// TIA Portal project "MAIN-PLS-AHS-100125" (V19)

(* hardware
DEVICE "S7-1200 station_1"  S7-1200 Station
   slot 0: "Rack_0"  S7-1200 Rack  Rack  V1.0
   slot 1: "PLC_1"  CPU 1214C AC/DC/Rly  6ES7 214-1BG40-0XB0  V4.6
DEVICE "ET 200SP station_1"  ET 200SP-Station
   slot 0: "Rack_0"  Rack  6ES5 710-8MAx1
   slot 0: "et200sp_greider"  IM 155-6 PN HF  6ES7 155-6AU00-0CN0  V4.2
   slot 1: "DI 8x24VDC HF_1"  DI 8x24VDC HF  6ES7 131-6BF00-0CA0  V2.0
      slot 1: "DI 8x24VDC HF_1"  DI 8x24VDC HF
   slot 2: "DI 8x24VDC HF_2"  DI 8x24VDC HF  6ES7 131-6BF00-0CA0  V2.0
      slot 1: "DI 8x24VDC HF_2"  DI 8x24VDC HF
   slot 3: "DI 8x24VDC HF_3"  DI 8x24VDC HF  6ES7 131-6BF00-0CA0  V2.0
      slot 1: "DI 8x24VDC HF_3"  DI 8x24VDC HF
   slot 4: "DI 8x24VDC HF_4"  DI 8x24VDC HF  6ES7 131-6BF00-0CA0  V2.0
      slot 1: "DI 8x24VDC HF_4"  DI 8x24VDC HF
   slot 5: "DQ 8x24VDC/0.5A HF_1"  DQ 8x24VDC/0.5A HF  6ES7 132-6BF00-0CA0  V2.0
      slot 1: "DQ 8x24VDC/0.5A HF_1"  DQ 8x24VDC/0.5A HF
   slot 6: "DQ 8x24VDC/0.5A HF_2"  DQ 8x24VDC/0.5A HF  6ES7 132-6BF00-0CA0  V2.0
      slot 1: "DQ 8x24VDC/0.5A HF_2"  DQ 8x24VDC/0.5A HF
   slot 7: "DQ 8x24VDC/0.5A HF_3"  DQ 8x24VDC/0.5A HF  6ES7 132-6BF00-0CA0  V2.0
      slot 1: "DQ 8x24VDC/0.5A HF_3"  DQ 8x24VDC/0.5A HF
   slot 8: "DQ 8x24VDC/0.5A HF_4"  DQ 8x24VDC/0.5A HF  6ES7 132-6BF00-0CA0  V2.0
      slot 1: "DQ 8x24VDC/0.5A HF_4"  DQ 8x24VDC/0.5A HF
   slot 9: "Server module_1"  Server module  6ES7 193-6PA00-0AA0  V1.1
      slot 1: "Server module_1"  Server module
   slot 127: "BA 2xRJ45"  BA 2xRJ45  6ES7 193-6AR00-0AA0  V0.0
      slot 1: "Port_1"  X1 P1 R  6ES7 193-6AR00-0AA0  V0.0
      slot 2: "Port_2"  X1 P2 R  6ES7 193-6AR00-0AA0  V0.0
DEVICE "ET 200SP station_2"  ET 200SP-Station
   slot 0: "Rack_0"  Rack  6ES5 710-8MAx1
   slot 0: "et200sp_servo"  IM 155-6 PN HF  6ES7 155-6AU00-0CN0  V4.2
   slot 1: "DI 8x24VDC HF_1"  DI 8x24VDC HF  6ES7 131-6BF00-0CA0  V2.0
      slot 1: "DI 8x24VDC HF_1"  DI 8x24VDC HF
   slot 2: "DI 8x24VDC HF_2"  DI 8x24VDC HF  6ES7 131-6BF00-0CA0  V2.0
      slot 1: "DI 8x24VDC HF_2"  DI 8x24VDC HF
   slot 3: "DQ 8x24VDC/0.5A HF_1"  DQ 8x24VDC/0.5A HF  6ES7 132-6BF00-0CA0  V2.0
      slot 1: "DQ 8x24VDC/0.5A HF_1"  DQ 8x24VDC/0.5A HF
   slot 4: "DQ 8x24VDC/0.5A HF_2"  DQ 8x24VDC/0.5A HF  6ES7 132-6BF00-0CA0  V2.0
      slot 1: "DQ 8x24VDC/0.5A HF_2"  DQ 8x24VDC/0.5A HF
   slot 5: "Server module_1"  Server module  6ES7 193-6PA00-0AA0  V1.1
      slot 1: "Server module_1"  Server module
   slot 127: "BA 2xRJ45"  BA 2xRJ45  6ES7 193-6AR00-0AA0  V0.0
      slot 1: "Port_1"  X1 P1 R  6ES7 193-6AR00-0AA0  V0.0
      slot 2: "Port_2"  X1 P2 R  6ES7 193-6AR00-0AA0  V0.0
*)

// ===== PLC "PLC_1"  CPU 1214C AC/DC/Rly =====

VAR_GLOBAL   // PLC tag table "Default tag table"
   "C1.1_I" AT %I2.0 : Bool;
   "C1.2_I" AT %I2.1 : Bool;
   "C2.1_I" AT %I2.2 : Bool;
   "C2.2_I" AT %I2.3 : Bool;
   "C3.1_I" AT %I2.4 : Bool;
   "C3.2_I" AT %I2.5 : Bool;
   "Fotocelle_I" AT %I2.6 : Bool;
   "A_IG_I" AT %I3.1 : Bool;
   "B_IG_I" AT %I3.2 : Bool;
   "Bryter_S1_Ved_HMI_I" AT %I0.0 : Bool;
   "Bryter_S5_Ved_HMI_I" AT %I0.4 : Bool;
   "Bryter_Høyre_Skap_I" AT %I3.3 : Bool;
   "Bryter_Venstre_Skap_I" AT %I3.4 : Bool;
   "Tag_10" AT %IW64 : Word;
   "Bryter_S2_Ved_HMI_I" AT %I0.1 : Bool;
   "Bryter_3_Ved_HMI_I" AT %I0.2 : Bool;
   "Bryter_S4_Ved_HMI_I" AT %I0.3 : Bool;
   "Tag_2" AT %I3.0 : Bool;
   "A-IG" AT %I4.0 : Bool;
   "16cm_Nærhetsføler_ved_robot" AT %I5.5 : Bool;
   "8cm_Nærhetsføler_ved_robot" AT %I5.6 : Bool;
   "Tag_7" AT %I5.7 : Bool;
   "12cm_Nærhetsføler_ved_robot" AT %I5.4 : Bool;
   "12_CM_Sluppet" AT %I5.1 : Bool;
   "8_CM_Sluppet" AT %I5.2 : Bool;
   "16_CM_Sluppet" AT %I5.3 : Bool;
   "16cm_knapp_main_skap" AT %I0.5 : Bool;
   "12cm_plukk_robot" AT %Q2.0 : Bool;
   "16cm_plukk_robot" AT %Q2.1 : Bool;
   "8_plukk_robot" AT %Q2.2 : Bool;
   "V2" AT %Q3.1 : Bool;
   "V1" AT %Q3.0 : Bool;
   "Tag_14" AT %Q0.2 : Bool;
   "V3" AT %Q3.2 : Bool;
   "C3" AT %Q3.3 : Bool;
   "Tag_9" AT %Q3.4 : Bool;
   "Tag_11" AT %QW68 : Word;
   "Tag_1" AT %QW70 : Word;
   "V4_Utgang" AT %Q4.0 : Bool;
   "V5_Utgang" AT %Q4.1 : Bool;
   "V6_Utgang" AT %Q4.2 : Bool;
   "C1.1_M" AT %M0.0 : Bool;
   "C1.2_M" AT %M0.1 : Bool;
   "C2.1_M" AT %M0.2 : Bool;
   "C2.2_M" AT %M0.3 : Bool;
   "C3.1_M" AT %M0.4 : Bool;
   "C3.2_M" AT %M0.5 : Bool;
   "Fotocelle_M" AT %M0.6 : Bool;
   "A_IG_M" AT %M0.7 : Bool;
   "Bryter_Høyre_Skap_M" AT %M1.1 : Bool;
   "B_IG_M" AT %M1.0 : Bool;
   "Bryter_S1_Ved_HMI_M" AT %M2.0 : Bool;
   "Bryter_S2_Ved_HMI_M" AT %M2.1 : Bool;
   "Bryter_S3_Ved_HMI_M" AT %M2.2 : Bool;
   "System_Byte" AT %MB8001 : Byte;
   "FirstScan" AT %M8001.0 : Bool;
   "DiagStatusUpdate" AT %M8001.1 : Bool;
   "AlwaysTRUE" AT %M8001.2 : Bool;
   "AlwaysFALSE" AT %M8001.3 : Bool;
   "Clock_Byte" AT %MB8000 : Byte;
   "Clock_10Hz" AT %M8000.0 : Bool;
   "Clock_5Hz" AT %M8000.1 : Bool;
   "Clock_2.5Hz" AT %M8000.2 : Bool;
   "Clock_2Hz" AT %M8000.3 : Bool;
   "Clock_1.25Hz" AT %M8000.4 : Bool;
   "Clock_1Hz" AT %M8000.5 : Bool;
   "Clock_0.625Hz" AT %M8000.6 : Bool;
   "Clock_0.5Hz" AT %M8000.7 : Bool;
   "Kloss1_8cm" AT %M10.0 : Bool;
   "delay_set_10.2" AT %M10.1 : Bool;
   "Kloss2_8cm" AT %M10.2 : Bool;
   "Tag_8" AT %M20.1 : Bool;
   "V1_Kloss1_U" AT %M11.0 : Bool;
   "V1_Kloss2_U" AT %M11.1 : Bool;
   "delay_set_10.4" AT %M10.3 : Bool;
   "Kloss3_8cm" AT %M10.4 : Bool;
   "V1_Kloss3_U" AT %M11.2 : Bool;
   "Kloss1_12cm" AT %M12.0 : Bool;
   "Kloss2_12cm" AT %M12.2 : Bool;
   "Kloss3_12cm" AT %M12.4 : Bool;
   "delay_set_12.4" AT %M12.3 : Bool;
   "delay_set_12.2" AT %M12.1 : Bool;
   "V2_Kloss2_U" AT %M13.1 : Bool;
   "V2_Kloss3_U" AT %M13.2 : Bool;
   "V2_Kloss1_U" AT %M13.0 : Bool;
   "Kloss4_12cm" AT %M12.6 : Bool;
   "delay_set_12.6" AT %M12.5 : Bool;
   "V2_Kloss4_U" AT %M13.3 : Bool;
   "delay_set_14.2" AT %M14.1 : Bool;
   "delay_set_14.4" AT %M14.3 : Bool;
   "delay_set_14.6" AT %M14.5 : Bool;
   "Kloss4_16cm" AT %M14.6 : Bool;
   "Kloss1_16cm" AT %M14.0 : Bool;
   "Kloss2_16cm" AT %M14.2 : Bool;
   "Kloss3_16cm" AT %M14.4 : Bool;
   "delay_set_15.0" AT %M14.7 : Bool;
   "Kloss5_16cm" AT %M15.0 : Bool;
   "V3_Kloss1_U" AT %M15.1 : Bool;
   "V3_Kloss2_U" AT %M15.2 : Bool;
   "V3_Kloss3_U" AT %M15.3 : Bool;
   "V3_Kloss4_U" AT %M15.4 : Bool;
   "V3_Kloss5_U" AT %M15.5 : Bool;
   "Bryter_Venstre_Skap_M" AT %M1.2 : Bool;
   "Bryter_S4_Ved_HMI_M" AT %M2.3 : Bool;
   "Bryter_S5_Ved_HMI_M" AT %M2.4 : Bool;
   "Ventil_4_UT" AT %M50.0 : Bool;
   "Ventil_5_UT" AT %M50.1 : Bool;
   "Ventil_6_UT" AT %M50.2 : Bool;
   "16CM_Pall_Full" AT %M5.0 : Bool;
   "12CM_Pall_Full" AT %M5.1 : Bool;
   "8CM_Pall_Full" AT %M5.2 : Bool;
   "Tag_15" AT %I3.5 : Bool;
   "Hent_8cm_til_Servo_Q" AT %Q6.0 : Bool;
   "Hent_12cm_til_Servo_Q" AT %Q6.1 : Bool;
   "Hent_16cm_til_Servo_Q" AT %Q6.2 : Bool;
   "Lever_12cm_til_servo_Q" AT %Q6.4 : Bool;
   "Lever_8cm_til_servo_Q" AT %Q6.5 : Bool;
   "Lever_16cm_til_servo_Q" AT %Q6.6 : Bool;
   "Ved_HentPos8cm_fra_servo" AT %I6.0 : Bool;
   "Ved_hentPos12cm_fra_servo" AT %I6.1 : Bool;
   "Ved_hentPos16cm_fra_servo" AT %I6.2 : Bool;
   "C4_PlussPos_I" AT %I4.1 : Bool;
   "C4_MinPos_I" AT %I4.2 : Bool;
   "C5_PlussPos_I" AT %I4.3 : Bool;
   "C5_MinPos_I" AT %I4.4 : Bool;
   "C6_PlussPos_I" AT %I4.5 : Bool;
   "C6_MinPos_I" AT %I4.6 : Bool;
   "C4_Retur_Set" AT %M51.0 : Bool;
   "Tag_3" AT %M1000.0 : Bool;
   "8cm_Pall_På_Plass" AT %M52.0 : Bool;
   "Bekreftet_levert_pall_16cm_fra_servo" AT %I6.5 : Bool;
   "Bekreftet_levering_8_cm_fra_servo" AT %I6.3 : Bool;
   "Vent_ny_pall_8cm" AT %M52.1 : Bool;
   "Vent_ny_pall_16cm" AT %M60.0 : Bool;
   "Tag_4" AT %I0.6 : Bool;
   "16cm_pall_på_plass" AT %M60.1 : Bool;
   "C6_retur_set" AT %M60.3 : Bool;
   "tag" AT %M60.2 : Bool;
END_VAR

// folder: System blocks/Program resources

DATA_BLOCK "300ms delay utskyt"   // DB1
{ S7_Optimized_Access := 'TRUE' }
AUTHOR : Simatic
FAMILY : IEC
NAME : IEC_TMR
VERSION : 1.0
// stored: InstanceOfName IEC_TIMER
"IEC_TIMER"
BEGIN
END_DATA_BLOCK

DATA_BLOCK "KLoss2_8cm_Husk_V1"   // DB2
{ S7_Optimized_Access := 'TRUE' }
AUTHOR : Simatic
FAMILY : IEC
NAME : CNTR
VERSION : 1.0
// stored: InstanceOfName IEC_COUNTER
"IEC_COUNTER"
BEGIN
END_DATA_BLOCK

DATA_BLOCK "300ms delay utskyt kloss2"   // DB3
{ S7_Optimized_Access := 'TRUE' }
AUTHOR : Simatic
FAMILY : IEC
NAME : IEC_TMR
VERSION : 1.0
// stored: InstanceOfName IEC_TIMER
"IEC_TIMER"
BEGIN
END_DATA_BLOCK

DATA_BLOCK "Klossestørrelse"   // DB4
{ S7_Optimized_Access := 'TRUE' }
AUTHOR : Simatic
FAMILY : IEC
NAME : CNTR
VERSION : 1.0
// stored: InstanceOfName IEC_COUNTER
"IEC_COUNTER"
BEGIN
END_DATA_BLOCK

DATA_BLOCK "250ms delay reset db4"   // DB5
{ S7_Optimized_Access := 'TRUE' }
AUTHOR : Simatic
FAMILY : IEC
NAME : IEC_TMR
VERSION : 1.0
// stored: InstanceOfName IEC_TIMER
"IEC_TIMER"
BEGIN
END_DATA_BLOCK

DATA_BLOCK "delay_set_m10.2"   // DB6
{ S7_Optimized_Access := 'TRUE' }
AUTHOR : Simatic
FAMILY : IEC
NAME : IEC_TMR
VERSION : 1.0
// stored: InstanceOfName IEC_TIMER
"IEC_TIMER"
BEGIN
END_DATA_BLOCK

DATA_BLOCK "Kloss1_Husk_V1"   // DB7
{ S7_Optimized_Access := 'TRUE' }
AUTHOR : Simatic
FAMILY : IEC
NAME : CNTR
VERSION : 1.0
// stored: InstanceOfName IEC_COUNTER
"IEC_COUNTER"
BEGIN
END_DATA_BLOCK

DATA_BLOCK "delay_inrange_reset"   // DB8
{ S7_Optimized_Access := 'TRUE' }
AUTHOR : Simatic
FAMILY : IEC
NAME : IEC_TMR
VERSION : 1.0
// stored: InstanceOfName IEC_TIMER
"IEC_TIMER"
BEGIN
END_DATA_BLOCK

DATA_BLOCK "delay_set_m10.4"   // DB9
{ S7_Optimized_Access := 'TRUE' }
AUTHOR : Simatic
FAMILY : IEC
NAME : IEC_TMR
VERSION : 1.0
// stored: InstanceOfName IEC_TIMER
"IEC_TIMER"
BEGIN
END_DATA_BLOCK

DATA_BLOCK "Kloss3_8cm_Husk_V1"   // DB10
{ S7_Optimized_Access := 'TRUE' }
AUTHOR : Simatic
FAMILY : IEC
NAME : CNTR
VERSION : 1.0
// stored: InstanceOfName IEC_COUNTER
"IEC_COUNTER"
BEGIN
END_DATA_BLOCK

DATA_BLOCK "300ms delay utskyt kloss3"   // DB11
{ S7_Optimized_Access := 'TRUE' }
AUTHOR : Simatic
FAMILY : IEC
NAME : IEC_TMR
VERSION : 1.0
// stored: InstanceOfName IEC_TIMER
"IEC_TIMER"
BEGIN
END_DATA_BLOCK

DATA_BLOCK "delay_inrange12cm_reset"   // DB12
{ S7_Optimized_Access := 'TRUE' }
AUTHOR : Simatic
FAMILY : IEC
NAME : IEC_TMR
VERSION : 1.0
// stored: InstanceOfName IEC_TIMER
"IEC_TIMER"
BEGIN
END_DATA_BLOCK

DATA_BLOCK "delay_set_m12.2"   // DB13
{ S7_Optimized_Access := 'TRUE' }
AUTHOR : Simatic
FAMILY : IEC
NAME : IEC_TMR
VERSION : 1.0
// stored: InstanceOfName IEC_TIMER
"IEC_TIMER"
BEGIN
END_DATA_BLOCK

DATA_BLOCK "delay_set_m12.4"   // DB14
{ S7_Optimized_Access := 'TRUE' }
AUTHOR : Simatic
FAMILY : IEC
NAME : IEC_TMR
VERSION : 1.0
// stored: InstanceOfName IEC_TIMER
"IEC_TIMER"
BEGIN
END_DATA_BLOCK

DATA_BLOCK "Kloss1_12cm_Husk_V2"   // DB15
{ S7_Optimized_Access := 'TRUE' }
AUTHOR : Simatic
FAMILY : IEC
NAME : CNTR
VERSION : 1.0
// stored: InstanceOfName IEC_COUNTER
"IEC_COUNTER"
BEGIN
END_DATA_BLOCK

DATA_BLOCK "Kloss2_12cm_Husk_V2"   // DB16
{ S7_Optimized_Access := 'TRUE' }
AUTHOR : Simatic
FAMILY : IEC
NAME : CNTR
VERSION : 1.0
// stored: InstanceOfName IEC_COUNTER
"IEC_COUNTER"
BEGIN
END_DATA_BLOCK

DATA_BLOCK "Kloss3_12cm_Husk_V2"   // DB17
{ S7_Optimized_Access := 'TRUE' }
AUTHOR : Simatic
FAMILY : IEC
NAME : CNTR
VERSION : 1.0
// stored: InstanceOfName IEC_COUNTER
"IEC_COUNTER"
BEGIN
END_DATA_BLOCK

DATA_BLOCK "300ms delay utskyt kloss1_12cm"   // DB18
{ S7_Optimized_Access := 'TRUE' }
AUTHOR : Simatic
FAMILY : IEC
NAME : IEC_TMR
VERSION : 1.0
// stored: InstanceOfName IEC_TIMER
"IEC_TIMER"
BEGIN
END_DATA_BLOCK

DATA_BLOCK "300ms delay utskyt kloss2_12cm"   // DB19
{ S7_Optimized_Access := 'TRUE' }
AUTHOR : Simatic
FAMILY : IEC
NAME : IEC_TMR
VERSION : 1.0
// stored: InstanceOfName IEC_TIMER
"IEC_TIMER"
BEGIN
END_DATA_BLOCK

DATA_BLOCK "300ms delay utskyt kloss3_12cm"   // DB20
{ S7_Optimized_Access := 'TRUE' }
AUTHOR : Simatic
FAMILY : IEC
NAME : IEC_TMR
VERSION : 1.0
// stored: InstanceOfName IEC_TIMER
"IEC_TIMER"
BEGIN
END_DATA_BLOCK

DATA_BLOCK "delay_set_m12.6"   // DB21
{ S7_Optimized_Access := 'TRUE' }
AUTHOR : Simatic
FAMILY : IEC
NAME : IEC_TMR
VERSION : 1.0
// stored: InstanceOfName IEC_TIMER
"IEC_TIMER"
BEGIN
END_DATA_BLOCK

DATA_BLOCK "Kloss4_12cm_Husk_V2"   // DB22
{ S7_Optimized_Access := 'TRUE' }
AUTHOR : Simatic
FAMILY : IEC
NAME : CNTR
VERSION : 1.0
// stored: InstanceOfName IEC_COUNTER
"IEC_COUNTER"
BEGIN
END_DATA_BLOCK

DATA_BLOCK "delay_inrange16cm_reset"   // DB23
{ S7_Optimized_Access := 'TRUE' }
AUTHOR : Simatic
FAMILY : IEC
NAME : IEC_TMR
VERSION : 1.0
// stored: InstanceOfName IEC_TIMER
"IEC_TIMER"
BEGIN
END_DATA_BLOCK

DATA_BLOCK "300ms delay utskyt kloss4_12cmTON"   // DB24
{ S7_Optimized_Access := 'TRUE' }
AUTHOR : Simatic
FAMILY : IEC
NAME : IEC_TMR
VERSION : 1.0
// stored: InstanceOfName IEC_TIMER
"IEC_TIMER"
BEGIN
END_DATA_BLOCK

DATA_BLOCK "delay_set_m14.2"   // DB25
{ S7_Optimized_Access := 'TRUE' }
AUTHOR : Simatic
FAMILY : IEC
NAME : IEC_TMR
VERSION : 1.0
// stored: InstanceOfName IEC_TIMER
"IEC_TIMER"
BEGIN
END_DATA_BLOCK

DATA_BLOCK "delay_set_m14.4"   // DB26
{ S7_Optimized_Access := 'TRUE' }
AUTHOR : Simatic
FAMILY : IEC
NAME : IEC_TMR
VERSION : 1.0
// stored: InstanceOfName IEC_TIMER
"IEC_TIMER"
BEGIN
END_DATA_BLOCK

DATA_BLOCK "delay_set_m14.6"   // DB27
{ S7_Optimized_Access := 'TRUE' }
AUTHOR : Simatic
FAMILY : IEC
NAME : IEC_TMR
VERSION : 1.0
// stored: InstanceOfName IEC_TIMER
"IEC_TIMER"
BEGIN
END_DATA_BLOCK

DATA_BLOCK "delay_set_m15.0"   // DB28
{ S7_Optimized_Access := 'TRUE' }
AUTHOR : Simatic
FAMILY : IEC
NAME : IEC_TMR
VERSION : 1.0
// stored: InstanceOfName IEC_TIMER
"IEC_TIMER"
BEGIN
END_DATA_BLOCK

DATA_BLOCK "Kloss5_16cm_Husk_V3"   // DB29
{ S7_Optimized_Access := 'TRUE' }
AUTHOR : Simatic
FAMILY : IEC
NAME : CNTR
VERSION : 1.0
// stored: InstanceOfName IEC_COUNTER
"IEC_COUNTER"
BEGIN
END_DATA_BLOCK

DATA_BLOCK "300ms delay utskyt kloss5_16cm"   // DB30
{ S7_Optimized_Access := 'TRUE' }
AUTHOR : Simatic
FAMILY : IEC
NAME : IEC_TMR
VERSION : 1.0
// stored: InstanceOfName IEC_TIMER
"IEC_TIMER"
BEGIN
END_DATA_BLOCK

DATA_BLOCK "Kloss1_16cm_Husk_V3"   // DB31
{ S7_Optimized_Access := 'TRUE' }
AUTHOR : Simatic
FAMILY : IEC
NAME : CNTR
VERSION : 1.0
// stored: InstanceOfName IEC_COUNTER
"IEC_COUNTER"
BEGIN
END_DATA_BLOCK

DATA_BLOCK "Kloss2_16cm_Husk_V3"   // DB32
{ S7_Optimized_Access := 'TRUE' }
AUTHOR : Simatic
FAMILY : IEC
NAME : CNTR
VERSION : 1.0
// stored: InstanceOfName IEC_COUNTER
"IEC_COUNTER"
BEGIN
END_DATA_BLOCK

DATA_BLOCK "Kloss3_16cm_Husk_V3"   // DB33
{ S7_Optimized_Access := 'TRUE' }
AUTHOR : Simatic
FAMILY : IEC
NAME : CNTR
VERSION : 1.0
// stored: InstanceOfName IEC_COUNTER
"IEC_COUNTER"
BEGIN
END_DATA_BLOCK

DATA_BLOCK "Kloss4_16cm_Husk_V3"   // DB34
{ S7_Optimized_Access := 'TRUE' }
AUTHOR : Simatic
FAMILY : IEC
NAME : CNTR
VERSION : 1.0
// stored: InstanceOfName IEC_COUNTER
"IEC_COUNTER"
BEGIN
END_DATA_BLOCK

DATA_BLOCK "300ms delay utskyt kloss1_16cm"   // DB35
{ S7_Optimized_Access := 'TRUE' }
AUTHOR : Simatic
FAMILY : IEC
NAME : IEC_TMR
VERSION : 1.0
// stored: InstanceOfName IEC_TIMER
"IEC_TIMER"
BEGIN
END_DATA_BLOCK

DATA_BLOCK "300ms delay utskyt kloss2_16cm"   // DB36
{ S7_Optimized_Access := 'TRUE' }
AUTHOR : Simatic
FAMILY : IEC
NAME : IEC_TMR
VERSION : 1.0
// stored: InstanceOfName IEC_TIMER
"IEC_TIMER"
BEGIN
END_DATA_BLOCK

DATA_BLOCK "300ms delay utskut kloss3_16cm"   // DB37
{ S7_Optimized_Access := 'TRUE' }
AUTHOR : Simatic
FAMILY : IEC
NAME : IEC_TMR
VERSION : 1.0
// stored: InstanceOfName IEC_TIMER
"IEC_TIMER"
BEGIN
END_DATA_BLOCK

DATA_BLOCK "300ms delay utskyt kloss4_16cm"   // DB38
{ S7_Optimized_Access := 'TRUE' }
AUTHOR : Simatic
FAMILY : IEC
NAME : IEC_TMR
VERSION : 1.0
// stored: InstanceOfName IEC_TIMER
"IEC_TIMER"
BEGIN
END_DATA_BLOCK

DATA_BLOCK "8cm_antall_HMI"   // DB39
{ S7_Optimized_Access := 'TRUE' }
AUTHOR : Simatic
FAMILY : IEC
NAME : CNTR
VERSION : 1.0
// stored: InstanceOfName IEC_COUNTER
"IEC_COUNTER"
BEGIN
END_DATA_BLOCK

DATA_BLOCK "12cm_antall_HMI"   // DB40
{ S7_Optimized_Access := 'TRUE' }
AUTHOR : Simatic
FAMILY : IEC
NAME : CNTR
VERSION : 1.0
// stored: InstanceOfName IEC_COUNTER
"IEC_COUNTER"
BEGIN
END_DATA_BLOCK

DATA_BLOCK "16cm_antall_HMI"   // DB41
{ S7_Optimized_Access := 'TRUE' }
AUTHOR : Simatic
FAMILY : IEC
NAME : CNTR
VERSION : 1.0
// stored: InstanceOfName IEC_COUNTER
"IEC_COUNTER"
BEGIN
END_DATA_BLOCK

DATA_BLOCK "blæææ"   // DB42
{ S7_Optimized_Access := 'TRUE' }
AUTHOR : Simatic
FAMILY : IEC
NAME : CNTR
VERSION : 1.0
// stored: InstanceOfName IEC_COUNTER
"IEC_COUNTER"
BEGIN
END_DATA_BLOCK

DATA_BLOCK "Antall_Palletert_16CM"   // DB43
{ S7_Optimized_Access := 'TRUE' }
AUTHOR : Simatic
FAMILY : IEC
NAME : CNTR
VERSION : 1.0
// stored: InstanceOfName IEC_COUNTER
"IEC_COUNTER"
BEGIN
END_DATA_BLOCK

DATA_BLOCK "Antall_Palletert_12CM"   // DB44
{ S7_Optimized_Access := 'TRUE' }
AUTHOR : Simatic
FAMILY : IEC
NAME : CNTR
VERSION : 1.0
// stored: InstanceOfName IEC_COUNTER
"IEC_COUNTER"
BEGIN
END_DATA_BLOCK

DATA_BLOCK "Antall_Palletert_8CM"   // DB45
{ S7_Optimized_Access := 'TRUE' }
AUTHOR : Simatic
FAMILY : IEC
NAME : CNTR
VERSION : 1.0
// stored: InstanceOfName IEC_COUNTER
"IEC_COUNTER"
BEGIN
END_DATA_BLOCK

// folder: (top level)

FUNCTION "InputMinne" : Void   // FC1, LAD
{ S7_Optimized_Access := 'TRUE' }
VERSION : 0.1
BEGIN

REGION Network 1
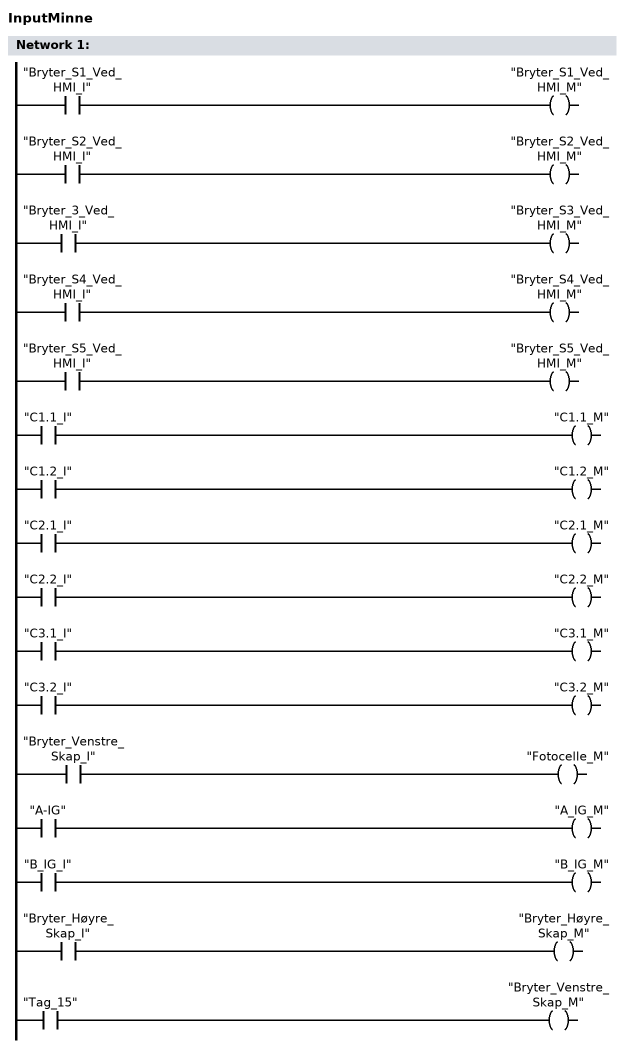
   RUNG wire#powerrail
      Contact( "Bryter_S1_Ved_HMI_I" )
      Coil( "Bryter_S1_Ved_HMI_M" )
   END_RUNG
   RUNG wire#powerrail
      Contact( "Bryter_S2_Ved_HMI_I" )
      Coil( "Bryter_S2_Ved_HMI_M" )
   END_RUNG
   RUNG wire#powerrail
      Contact( "Bryter_3_Ved_HMI_I" )
      Coil( "Bryter_S3_Ved_HMI_M" )
   END_RUNG
   RUNG wire#powerrail
      Contact( "Bryter_S4_Ved_HMI_I" )
      Coil( "Bryter_S4_Ved_HMI_M" )
   END_RUNG
   RUNG wire#powerrail
      Contact( "Bryter_S5_Ved_HMI_I" )
      Coil( "Bryter_S5_Ved_HMI_M" )
   END_RUNG
   RUNG wire#powerrail
      Contact( "C1.1_I" )
      Coil( "C1.1_M" )
   END_RUNG
   RUNG wire#powerrail
      Contact( "C1.2_I" )
      Coil( "C1.2_M" )
   END_RUNG
   RUNG wire#powerrail
      Contact( "C2.1_I" )
      Coil( "C2.1_M" )
   END_RUNG
   RUNG wire#powerrail
      Contact( "C2.2_I" )
      Coil( "C2.2_M" )
   END_RUNG
   RUNG wire#powerrail
      Contact( "C3.1_I" )
      Coil( "C3.1_M" )
   END_RUNG
   RUNG wire#powerrail
      Contact( "C3.2_I" )
      Coil( "C3.2_M" )
   END_RUNG
   RUNG wire#powerrail
      Contact( "Bryter_Venstre_Skap_I" )
      Coil( "Fotocelle_M" )
   END_RUNG
   RUNG wire#powerrail
      Contact( "A-IG" )
      Coil( "A_IG_M" )
   END_RUNG
   RUNG wire#powerrail
      Contact( "B_IG_I" )
      Coil( "B_IG_M" )
   END_RUNG
   RUNG wire#powerrail
      Contact( "Bryter_Høyre_Skap_I" )
      Coil( "Bryter_Høyre_Skap_M" )
   END_RUNG
   RUNG wire#powerrail
      Contact( "Tag_15" )
      Coil( "Bryter_Venstre_Skap_M" )
   END_RUNG
   // the same network as SCL:
   "Bryter_S1_Ved_HMI_M" := "Bryter_S1_Ved_HMI_I";
   "Bryter_S2_Ved_HMI_M" := "Bryter_S2_Ved_HMI_I";
   "Bryter_S3_Ved_HMI_M" := "Bryter_3_Ved_HMI_I";
   "Bryter_S4_Ved_HMI_M" := "Bryter_S4_Ved_HMI_I";
   "Bryter_S5_Ved_HMI_M" := "Bryter_S5_Ved_HMI_I";
   "C1.1_M" := "C1.1_I";
   "C1.2_M" := "C1.2_I";
   "C2.1_M" := "C2.1_I";
   "C2.2_M" := "C2.2_I";
   "C3.1_M" := "C3.1_I";
   "C3.2_M" := "C3.2_I";
   "Fotocelle_M" := "Bryter_Venstre_Skap_I";
   "A_IG_M" := "A-IG";
   "B_IG_M" := "B_IG_I";
   "Bryter_Høyre_Skap_M" := "Bryter_Høyre_Skap_I";
   "Bryter_Venstre_Skap_M" := "Tag_15";
END_REGION
END_FUNCTION

FUNCTION "GreiderStyring" : Void   // FC2, LAD
{ S7_Optimized_Access := 'TRUE' }
VERSION : 0.1
   VAR_TEMP   // added for the SCL form of the ladder/FBD networks
      _w1 : Bool;
   END_VAR
BEGIN

REGION Network 1
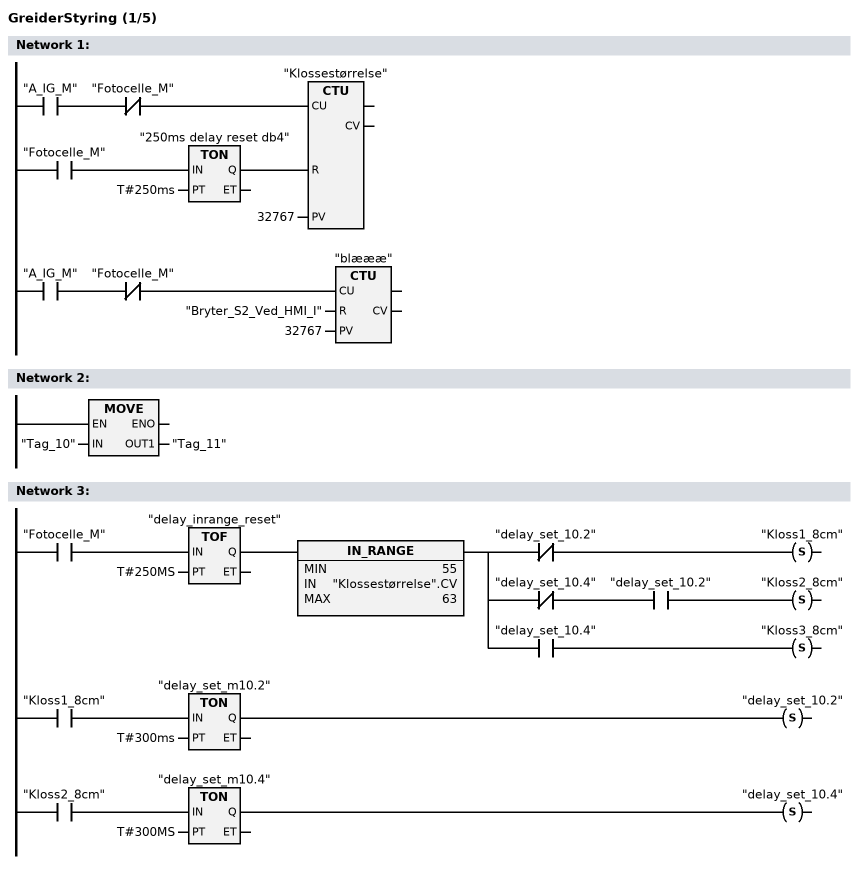
   "250ms delay reset db4".TON(IN := "Fotocelle_M", PT := T#250ms);
   "Klossestørrelse".CTU(CU := "A_IG_M" AND NOT "Fotocelle_M", R := "250ms delay reset db4".Q, PV := 32767);
   "blæææ".CTU(CU := "A_IG_M" AND NOT "Fotocelle_M", R := "Bryter_S2_Ved_HMI_I", PV := 32767);
END_REGION

REGION Network 2
   RUNG wire#powerrail
      Move(in := "Tag_10", out1 => "Tag_11")
   END_RUNG
   // the same network as SCL:
   "Tag_11" := "Tag_10";
END_REGION

REGION Network 3
   "delay_inrange_reset".TOF(IN := "Fotocelle_M", PT := T#250MS);
   #_w1 := "delay_inrange_reset".Q AND (55 <= "Klossestørrelse".CV) AND ("Klossestørrelse".CV <= 63);
   IF #_w1 AND NOT "delay_set_10.2" THEN "Kloss1_8cm" := TRUE; END_IF;
   IF #_w1 AND NOT "delay_set_10.4" AND "delay_set_10.2" THEN "Kloss2_8cm" := TRUE; END_IF;
   IF #_w1 AND "delay_set_10.4" THEN "Kloss3_8cm" := TRUE; END_IF;
   "delay_set_m10.2".TON(IN := "Kloss1_8cm", PT := T#300ms);
   IF "delay_set_m10.2".Q THEN "delay_set_10.2" := TRUE; END_IF;
   "delay_set_m10.4".TON(IN := "Kloss2_8cm", PT := T#300MS);
   IF "delay_set_m10.4".Q THEN "delay_set_10.4" := TRUE; END_IF;
END_REGION

REGION Network 4
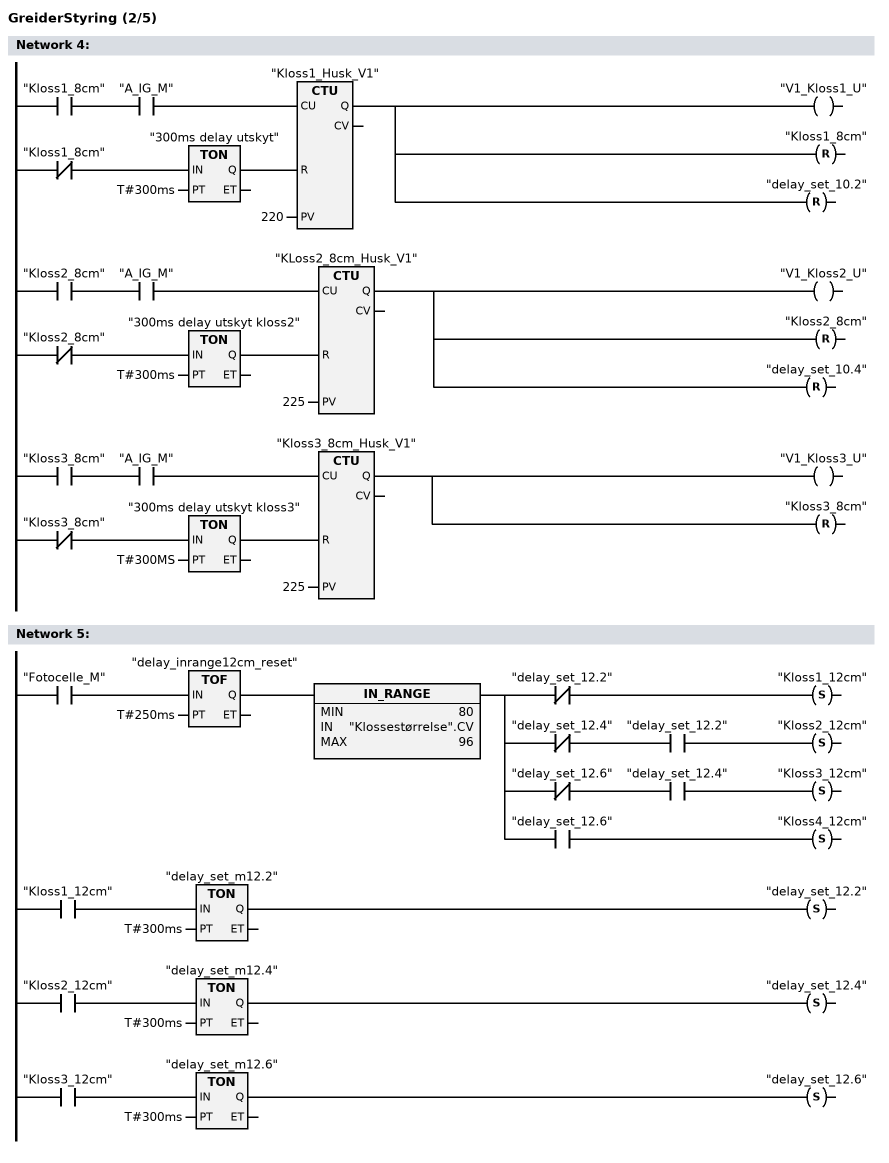
   "300ms delay utskyt".TON(IN := NOT "Kloss1_8cm", PT := T#300ms);
   "Kloss1_Husk_V1".CTU(CU := "Kloss1_8cm" AND "A_IG_M", R := "300ms delay utskyt".Q, PV := 220);
   "V1_Kloss1_U" := "Kloss1_Husk_V1".Q;
   IF "Kloss1_Husk_V1".Q THEN
       "Kloss1_8cm" := FALSE;
       "delay_set_10.2" := FALSE;
   END_IF;
   "300ms delay utskyt kloss2".TON(IN := NOT "Kloss2_8cm", PT := T#300ms);
   "KLoss2_8cm_Husk_V1".CTU(CU := "Kloss2_8cm" AND "A_IG_M", R := "300ms delay utskyt kloss2".Q, PV := 225);
   "V1_Kloss2_U" := "KLoss2_8cm_Husk_V1".Q;
   IF "KLoss2_8cm_Husk_V1".Q THEN
       "Kloss2_8cm" := FALSE;
       "delay_set_10.4" := FALSE;
   END_IF;
   "300ms delay utskyt kloss3".TON(IN := NOT "Kloss3_8cm", PT := T#300MS);
   "Kloss3_8cm_Husk_V1".CTU(CU := "Kloss3_8cm" AND "A_IG_M", R := "300ms delay utskyt kloss3".Q, PV := 225);
   "V1_Kloss3_U" := "Kloss3_8cm_Husk_V1".Q;
   IF "Kloss3_8cm_Husk_V1".Q THEN "Kloss3_8cm" := FALSE; END_IF;
END_REGION

REGION Network 5
   "delay_inrange12cm_reset".TOF(IN := "Fotocelle_M", PT := T#250ms);
   #_w1 := "delay_inrange12cm_reset".Q AND (80 <= "Klossestørrelse".CV) AND ("Klossestørrelse".CV <= 96);
   IF #_w1 AND NOT "delay_set_12.2" THEN "Kloss1_12cm" := TRUE; END_IF;
   IF #_w1 AND NOT "delay_set_12.4" AND "delay_set_12.2" THEN "Kloss2_12cm" := TRUE; END_IF;
   IF #_w1 AND NOT "delay_set_12.6" AND "delay_set_12.4" THEN "Kloss3_12cm" := TRUE; END_IF;
   IF #_w1 AND "delay_set_12.6" THEN "Kloss4_12cm" := TRUE; END_IF;
   "delay_set_m12.2".TON(IN := "Kloss1_12cm", PT := T#300ms);
   IF "delay_set_m12.2".Q THEN "delay_set_12.2" := TRUE; END_IF;
   "delay_set_m12.4".TON(IN := "Kloss2_12cm", PT := T#300ms);
   IF "delay_set_m12.4".Q THEN "delay_set_12.4" := TRUE; END_IF;
   "delay_set_m12.6".TON(IN := "Kloss3_12cm", PT := T#300ms);
   IF "delay_set_m12.6".Q THEN "delay_set_12.6" := TRUE; END_IF;
END_REGION

REGION Network 6
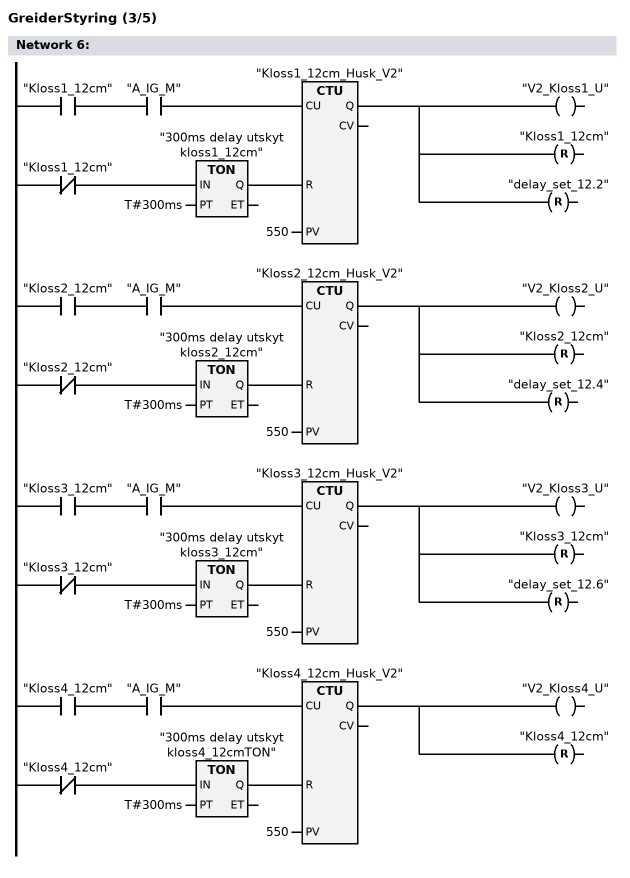
   "300ms delay utskyt kloss1_12cm".TON(IN := NOT "Kloss1_12cm", PT := T#300ms);
   "Kloss1_12cm_Husk_V2".CTU(CU := "Kloss1_12cm" AND "A_IG_M",
                           R := "300ms delay utskyt kloss1_12cm".Q,
                           PV := 550);
   "V2_Kloss1_U" := "Kloss1_12cm_Husk_V2".Q;
   IF "Kloss1_12cm_Husk_V2".Q THEN
       "Kloss1_12cm" := FALSE;
       "delay_set_12.2" := FALSE;
   END_IF;
   "300ms delay utskyt kloss2_12cm".TON(IN := NOT "Kloss2_12cm", PT := T#300ms);
   "Kloss2_12cm_Husk_V2".CTU(CU := "Kloss2_12cm" AND "A_IG_M",
                           R := "300ms delay utskyt kloss2_12cm".Q,
                           PV := 550);
   "V2_Kloss2_U" := "Kloss2_12cm_Husk_V2".Q;
   IF "Kloss2_12cm_Husk_V2".Q THEN
       "Kloss2_12cm" := FALSE;
       "delay_set_12.4" := FALSE;
   END_IF;
   "300ms delay utskyt kloss3_12cm".TON(IN := NOT "Kloss3_12cm", PT := T#300ms);
   "Kloss3_12cm_Husk_V2".CTU(CU := "Kloss3_12cm" AND "A_IG_M",
                           R := "300ms delay utskyt kloss3_12cm".Q,
                           PV := 550);
   "V2_Kloss3_U" := "Kloss3_12cm_Husk_V2".Q;
   IF "Kloss3_12cm_Husk_V2".Q THEN
       "Kloss3_12cm" := FALSE;
       "delay_set_12.6" := FALSE;
   END_IF;
   "300ms delay utskyt kloss4_12cmTON".TON(IN := NOT "Kloss4_12cm", PT := T#300ms);
   "Kloss4_12cm_Husk_V2".CTU(CU := "Kloss4_12cm" AND "A_IG_M",
                           R := "300ms delay utskyt kloss4_12cmTON".Q,
                           PV := 550);
   "V2_Kloss4_U" := "Kloss4_12cm_Husk_V2".Q;
   IF "Kloss4_12cm_Husk_V2".Q THEN "Kloss4_12cm" := FALSE; END_IF;
END_REGION

REGION Network 7
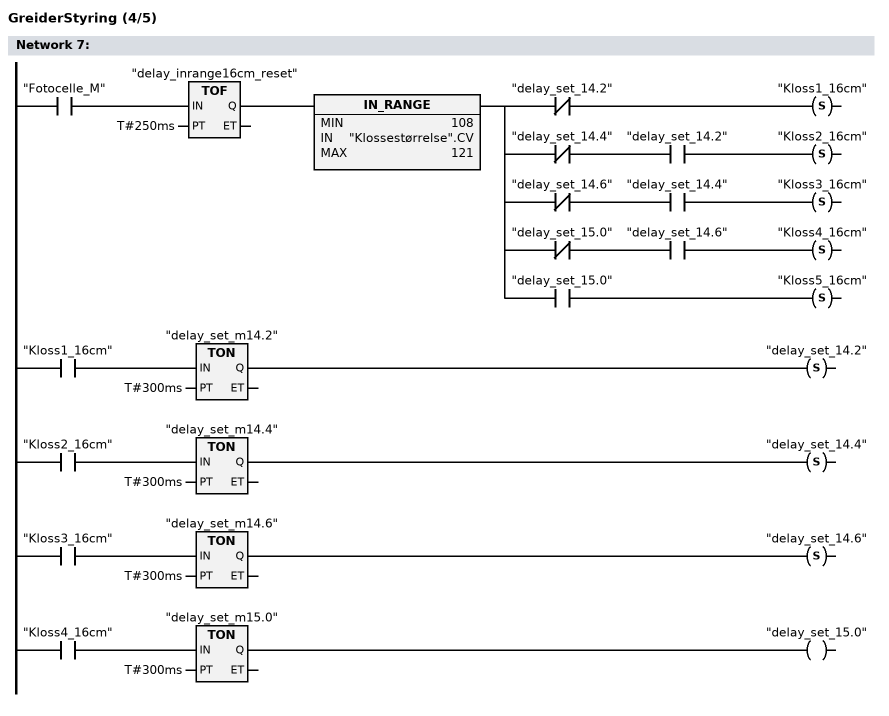
   "delay_inrange16cm_reset".TOF(IN := "Fotocelle_M", PT := T#250ms);
   #_w1 := "delay_inrange16cm_reset".Q AND (108 <= "Klossestørrelse".CV) AND ("Klossestørrelse".CV <= 121);
   IF #_w1 AND NOT "delay_set_14.2" THEN "Kloss1_16cm" := TRUE; END_IF;
   IF #_w1 AND NOT "delay_set_14.4" AND "delay_set_14.2" THEN "Kloss2_16cm" := TRUE; END_IF;
   IF #_w1 AND NOT "delay_set_14.6" AND "delay_set_14.4" THEN "Kloss3_16cm" := TRUE; END_IF;
   IF #_w1 AND NOT "delay_set_15.0" AND "delay_set_14.6" THEN "Kloss4_16cm" := TRUE; END_IF;
   IF #_w1 AND "delay_set_15.0" THEN "Kloss5_16cm" := TRUE; END_IF;
   "delay_set_m14.2".TON(IN := "Kloss1_16cm", PT := T#300ms);
   IF "delay_set_m14.2".Q THEN "delay_set_14.2" := TRUE; END_IF;
   "delay_set_m14.4".TON(IN := "Kloss2_16cm", PT := T#300ms);
   IF "delay_set_m14.4".Q THEN "delay_set_14.4" := TRUE; END_IF;
   "delay_set_m14.6".TON(IN := "Kloss3_16cm", PT := T#300ms);
   IF "delay_set_m14.6".Q THEN "delay_set_14.6" := TRUE; END_IF;
   "delay_set_m15.0".TON(IN := "Kloss4_16cm", PT := T#300ms);
   "delay_set_15.0" := "delay_set_m15.0".Q;
END_REGION

REGION Network 8
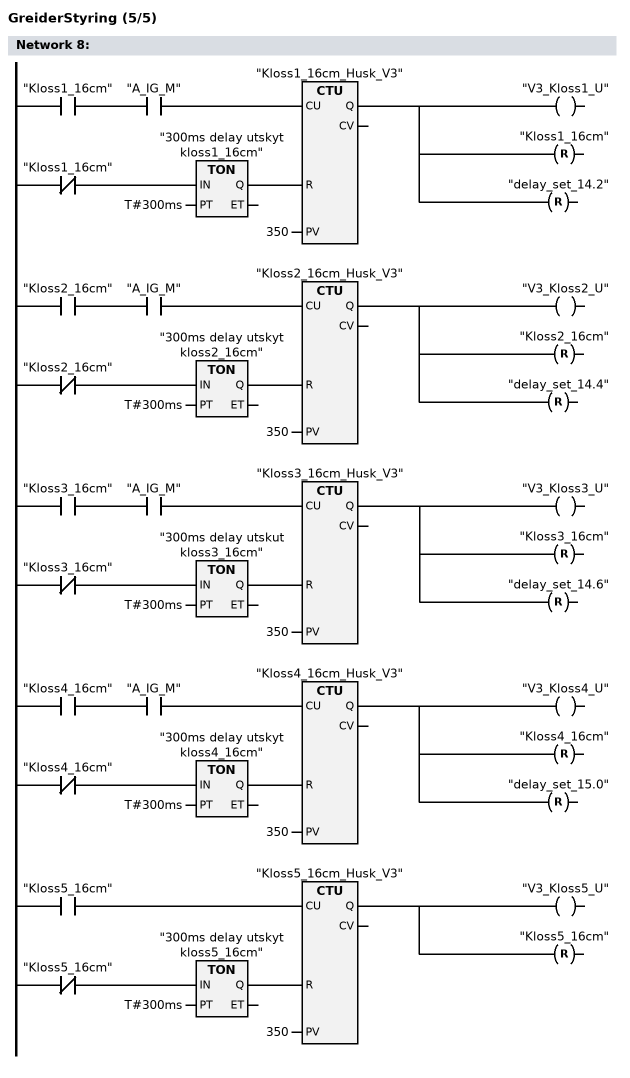
   "300ms delay utskyt kloss1_16cm".TON(IN := NOT "Kloss1_16cm", PT := T#300ms);
   "Kloss1_16cm_Husk_V3".CTU(CU := "Kloss1_16cm" AND "A_IG_M",
                           R := "300ms delay utskyt kloss1_16cm".Q,
                           PV := 350);
   "V3_Kloss1_U" := "Kloss1_16cm_Husk_V3".Q;
   IF "Kloss1_16cm_Husk_V3".Q THEN
       "Kloss1_16cm" := FALSE;
       "delay_set_14.2" := FALSE;
   END_IF;
   "300ms delay utskyt kloss2_16cm".TON(IN := NOT "Kloss2_16cm", PT := T#300ms);
   "Kloss2_16cm_Husk_V3".CTU(CU := "Kloss2_16cm" AND "A_IG_M",
                           R := "300ms delay utskyt kloss2_16cm".Q,
                           PV := 350);
   "V3_Kloss2_U" := "Kloss2_16cm_Husk_V3".Q;
   IF "Kloss2_16cm_Husk_V3".Q THEN
       "Kloss2_16cm" := FALSE;
       "delay_set_14.4" := FALSE;
   END_IF;
   "300ms delay utskut kloss3_16cm".TON(IN := NOT "Kloss3_16cm", PT := T#300ms);
   "Kloss3_16cm_Husk_V3".CTU(CU := "Kloss3_16cm" AND "A_IG_M",
                           R := "300ms delay utskut kloss3_16cm".Q,
                           PV := 350);
   "V3_Kloss3_U" := "Kloss3_16cm_Husk_V3".Q;
   IF "Kloss3_16cm_Husk_V3".Q THEN
       "Kloss3_16cm" := FALSE;
       "delay_set_14.6" := FALSE;
   END_IF;
   "300ms delay utskyt kloss4_16cm".TON(IN := NOT "Kloss4_16cm", PT := T#300ms);
   "Kloss4_16cm_Husk_V3".CTU(CU := "Kloss4_16cm" AND "A_IG_M",
                           R := "300ms delay utskyt kloss4_16cm".Q,
                           PV := 350);
   "V3_Kloss4_U" := "Kloss4_16cm_Husk_V3".Q;
   IF "Kloss4_16cm_Husk_V3".Q THEN
       "Kloss4_16cm" := FALSE;
       "delay_set_15.0" := FALSE;
   END_IF;
   "300ms delay utskyt kloss5_16cm".TON(IN := NOT "Kloss5_16cm", PT := T#300ms);
   "Kloss5_16cm_Husk_V3".CTU(CU := "Kloss5_16cm", R := "300ms delay utskyt kloss5_16cm".Q, PV := 350);
   "V3_Kloss5_U" := "Kloss5_16cm_Husk_V3".Q;
   IF "Kloss5_16cm_Husk_V3".Q THEN "Kloss5_16cm" := FALSE; END_IF;
END_REGION
END_FUNCTION

FUNCTION "Utgangskretser" : Void   // FC3, LAD
{ S7_Optimized_Access := 'TRUE' }
VERSION : 0.1
BEGIN

REGION Network 1
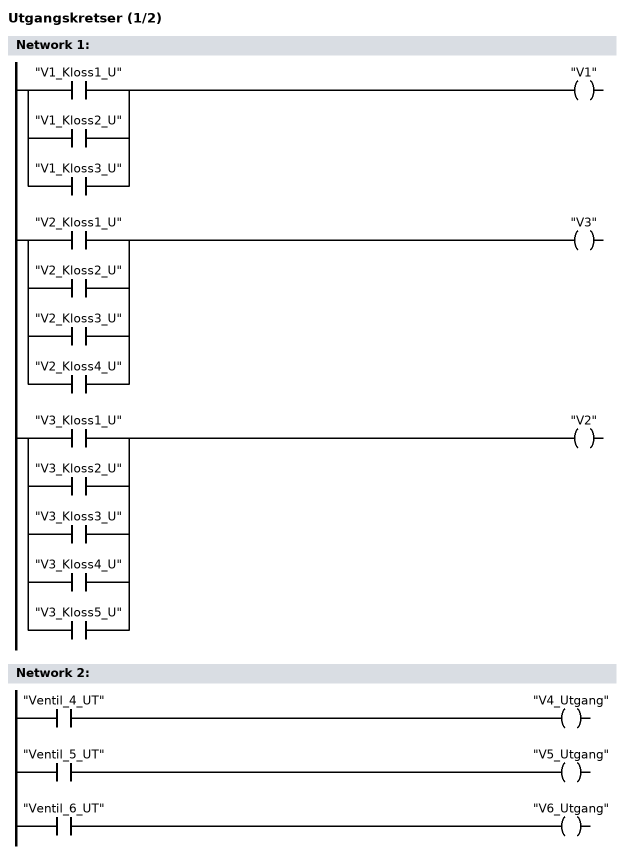
   RUNG wire#powerrail
      Contact( "V1_Kloss1_U" )
      wire#w1
      Coil( "V1" )
   END_RUNG
   RUNG wire#powerrail
      Contact( "V1_Kloss2_U" )
   END_RUNG wire#w1
   RUNG wire#powerrail
      Contact( "V1_Kloss3_U" )
   END_RUNG wire#w1
   RUNG wire#powerrail
      Contact( "V2_Kloss1_U" )
      wire#w2
      Coil( "V3" )
   END_RUNG
   RUNG wire#powerrail
      Contact( "V2_Kloss2_U" )
   END_RUNG wire#w2
   RUNG wire#powerrail
      Contact( "V2_Kloss3_U" )
   END_RUNG wire#w2
   RUNG wire#powerrail
      Contact( "V2_Kloss4_U" )
   END_RUNG wire#w2
   RUNG wire#powerrail
      Contact( "V3_Kloss1_U" )
      wire#w3
      Coil( "V2" )
   END_RUNG
   RUNG wire#powerrail
      Contact( "V3_Kloss2_U" )
   END_RUNG wire#w3
   RUNG wire#powerrail
      Contact( "V3_Kloss3_U" )
   END_RUNG wire#w3
   RUNG wire#powerrail
      Contact( "V3_Kloss4_U" )
   END_RUNG wire#w3
   RUNG wire#powerrail
      Contact( "V3_Kloss5_U" )
   END_RUNG wire#w3
   // the same network as SCL:
   "V1" := "V1_Kloss1_U" OR "V1_Kloss2_U" OR "V1_Kloss3_U";
   "V3" := "V2_Kloss1_U" OR "V2_Kloss2_U" OR "V2_Kloss3_U" OR "V2_Kloss4_U";
   "V2" := "V3_Kloss1_U" OR "V3_Kloss2_U" OR "V3_Kloss3_U" OR "V3_Kloss4_U" OR "V3_Kloss5_U";
END_REGION

REGION Network 2
   RUNG wire#powerrail
      Contact( "Ventil_4_UT" )
      Coil( "V4_Utgang" )
   END_RUNG
   RUNG wire#powerrail
      Contact( "Ventil_5_UT" )
      Coil( "V5_Utgang" )
   END_RUNG
   RUNG wire#powerrail
      Contact( "Ventil_6_UT" )
      Coil( "V6_Utgang" )
   END_RUNG
   // the same network as SCL:
   "V4_Utgang" := "Ventil_4_UT";
   "V5_Utgang" := "Ventil_5_UT";
   "V6_Utgang" := "Ventil_6_UT";
END_REGION

REGION Network 3
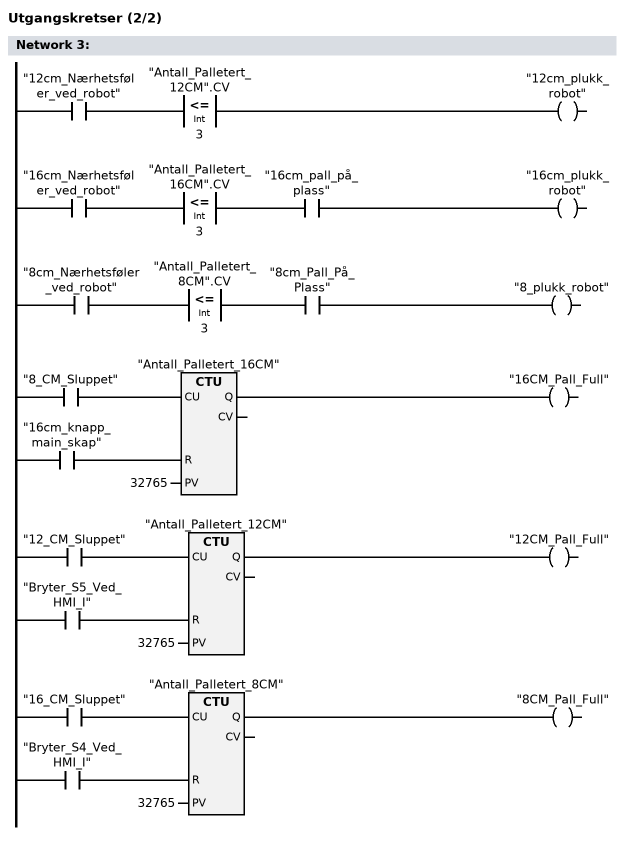
   "12cm_plukk_robot" := "12cm_Nærhetsføler_ved_robot" AND ("Antall_Palletert_12CM".CV <= 3);
   "16cm_plukk_robot" := "16cm_Nærhetsføler_ved_robot" AND ("Antall_Palletert_16CM".CV <= 3) AND "16cm_pall_på_plass";
   "8_plukk_robot" := "8cm_Nærhetsføler_ved_robot" AND ("Antall_Palletert_8CM".CV <= 3) AND "8cm_Pall_På_Plass";
   "Antall_Palletert_16CM".CTU(CU := "8_CM_Sluppet", R := "16cm_knapp_main_skap", PV := 32765);
   "16CM_Pall_Full" := "Antall_Palletert_16CM".Q;
   "Antall_Palletert_12CM".CTU(CU := "12_CM_Sluppet", R := "Bryter_S5_Ved_HMI_I", PV := 32765);
   "12CM_Pall_Full" := "Antall_Palletert_12CM".Q;
   "Antall_Palletert_8CM".CTU(CU := "16_CM_Sluppet", R := "Bryter_S4_Ved_HMI_I", PV := 32765);
   "8CM_Pall_Full" := "Antall_Palletert_8CM".Q;
END_REGION
END_FUNCTION

FUNCTION "HMI" : Void   // FC4, LAD
{ S7_Optimized_Access := 'TRUE' }
VERSION : 0.1
BEGIN

REGION Network 1
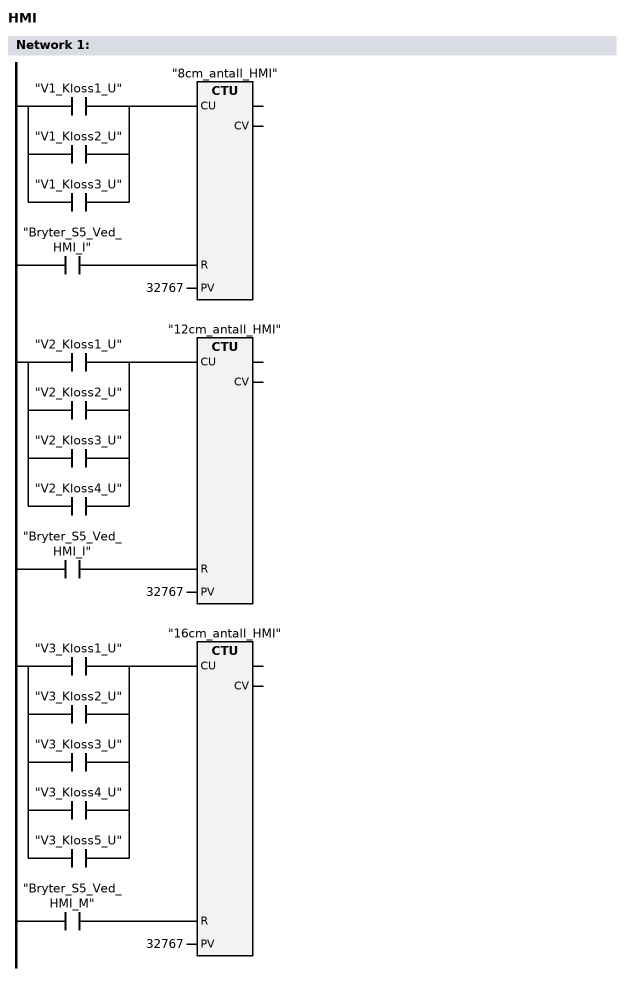
   "8cm_antall_HMI".CTU(CU := "V1_Kloss1_U" OR "V1_Kloss2_U" OR "V1_Kloss3_U",
                        R := "Bryter_S5_Ved_HMI_I",
                        PV := 32767);
   "12cm_antall_HMI".CTU(CU := "V2_Kloss1_U" OR "V2_Kloss2_U" OR "V2_Kloss3_U" OR "V2_Kloss4_U",
                         R := "Bryter_S5_Ved_HMI_I",
                         PV := 32767);
   "16cm_antall_HMI".CTU(CU := "V3_Kloss1_U" OR "V3_Kloss2_U" OR "V3_Kloss3_U" OR "V3_Kloss4_U" OR "V3_Kloss5_U",
                         R := "Bryter_S5_Ved_HMI_M",
                         PV := 32767);
END_REGION
END_FUNCTION

FUNCTION "Servo_PLS_Styring" : Void   // FC5, LAD
{ S7_Optimized_Access := 'TRUE' }
VERSION : 0.1
BEGIN

REGION Network 1
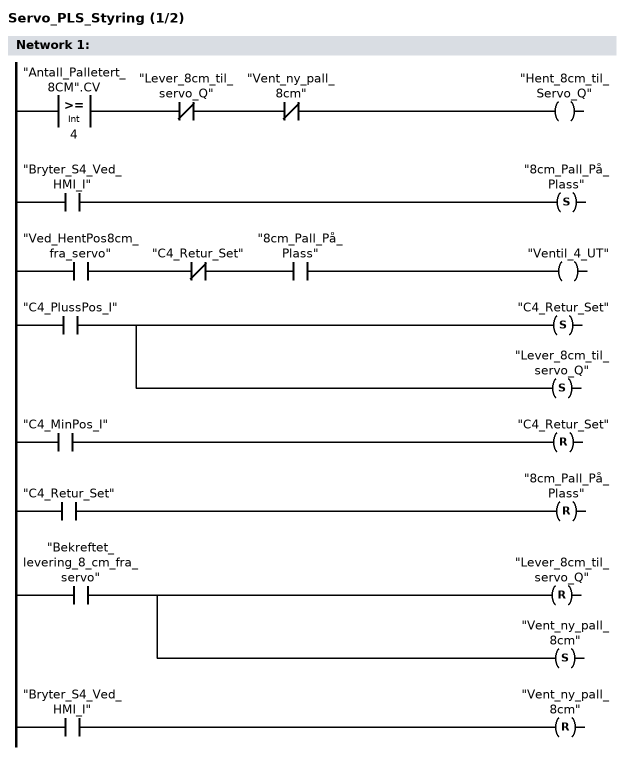
   RUNG wire#powerrail
      { S7_Templates := "SrcType := Int" } GE_Contact(in1 := "Antall_Palletert_8CM".CV, in2 := 4)
      I_Contact( "Lever_8cm_til_servo_Q" )
      I_Contact( "Vent_ny_pall_8cm" )
      Coil( "Hent_8cm_til_Servo_Q" )
   END_RUNG
   RUNG wire#powerrail
      Contact( "Bryter_S4_Ved_HMI_I" )
      S_Coil( "8cm_Pall_På_Plass" )
   END_RUNG
   RUNG wire#powerrail
      Contact( "Ved_HentPos8cm_fra_servo" )
      I_Contact( "C4_Retur_Set" )
      Contact( "8cm_Pall_På_Plass" )
      Coil( "Ventil_4_UT" )
   END_RUNG
   RUNG wire#powerrail
      Contact( "C4_PlussPos_I" )
      wire#w1
      S_Coil( "C4_Retur_Set" )
   END_RUNG
   RUNG wire#w1
      S_Coil( "Lever_8cm_til_servo_Q" )
   END_RUNG
   RUNG wire#powerrail
      Contact( "C4_MinPos_I" )
      R_Coil( "C4_Retur_Set" )
   END_RUNG
   RUNG wire#powerrail
      Contact( "C4_Retur_Set" )
      R_Coil( "8cm_Pall_På_Plass" )
   END_RUNG
   RUNG wire#powerrail
      Contact( "Bekreftet_levering_8_cm_fra_servo" )
      wire#w2
      R_Coil( "Lever_8cm_til_servo_Q" )
   END_RUNG
   RUNG wire#w2
      S_Coil( "Vent_ny_pall_8cm" )
   END_RUNG
   RUNG wire#powerrail
      Contact( "Bryter_S4_Ved_HMI_I" )
      R_Coil( "Vent_ny_pall_8cm" )
   END_RUNG
   // the same network as SCL:
   "Hent_8cm_til_Servo_Q" := ("Antall_Palletert_8CM".CV >= 4) AND NOT "Lever_8cm_til_servo_Q" AND NOT "Vent_ny_pall_8cm";
   IF "Bryter_S4_Ved_HMI_I" THEN "8cm_Pall_På_Plass" := TRUE; END_IF;
   "Ventil_4_UT" := "Ved_HentPos8cm_fra_servo" AND NOT "C4_Retur_Set" AND "8cm_Pall_På_Plass";
   IF "C4_PlussPos_I" THEN
       "C4_Retur_Set" := TRUE;
       "Lever_8cm_til_servo_Q" := TRUE;
   END_IF;
   IF "C4_MinPos_I" THEN "C4_Retur_Set" := FALSE; END_IF;
   IF "C4_Retur_Set" THEN "8cm_Pall_På_Plass" := FALSE; END_IF;
   IF "Bekreftet_levering_8_cm_fra_servo" THEN
       "Lever_8cm_til_servo_Q" := FALSE;
       "Vent_ny_pall_8cm" := TRUE;
   END_IF;
   IF "Bryter_S4_Ved_HMI_I" THEN "Vent_ny_pall_8cm" := FALSE; END_IF;
END_REGION

REGION Network 2
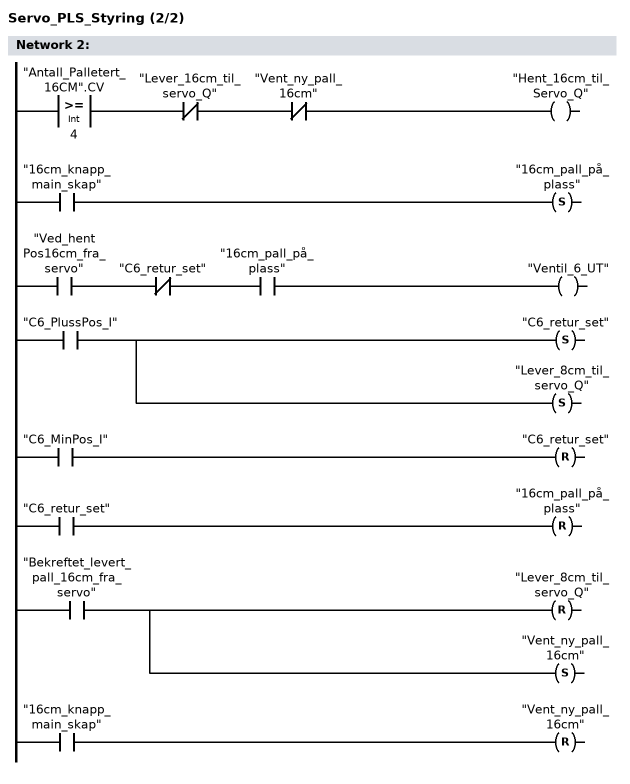
   RUNG wire#powerrail
      { S7_Templates := "SrcType := Int" } GE_Contact(in1 := "Antall_Palletert_16CM".CV, in2 := 4)
      I_Contact( "Lever_16cm_til_servo_Q" )
      I_Contact( "Vent_ny_pall_16cm" )
      Coil( "Hent_16cm_til_Servo_Q" )
   END_RUNG
   RUNG wire#powerrail
      Contact( "16cm_knapp_main_skap" )
      S_Coil( "16cm_pall_på_plass" )
   END_RUNG
   RUNG wire#powerrail
      Contact( "Ved_hentPos16cm_fra_servo" )
      I_Contact( "C6_retur_set" )
      Contact( "16cm_pall_på_plass" )
      Coil( "Ventil_6_UT" )
   END_RUNG
   RUNG wire#powerrail
      Contact( "C6_PlussPos_I" )
      wire#w1
      S_Coil( "C6_retur_set" )
   END_RUNG
   RUNG wire#w1
      S_Coil( "Lever_8cm_til_servo_Q" )
   END_RUNG
   RUNG wire#powerrail
      Contact( "C6_MinPos_I" )
      R_Coil( "C6_retur_set" )
   END_RUNG
   RUNG wire#powerrail
      Contact( "C6_retur_set" )
      R_Coil( "16cm_pall_på_plass" )
   END_RUNG
   RUNG wire#powerrail
      Contact( "Bekreftet_levert_pall_16cm_fra_servo" )
      wire#w2
      R_Coil( "Lever_8cm_til_servo_Q" )
   END_RUNG
   RUNG wire#w2
      S_Coil( "Vent_ny_pall_16cm" )
   END_RUNG
   RUNG wire#powerrail
      Contact( "16cm_knapp_main_skap" )
      R_Coil( "Vent_ny_pall_16cm" )
   END_RUNG
   // the same network as SCL:
   "Hent_16cm_til_Servo_Q" := ("Antall_Palletert_16CM".CV >= 4) AND NOT "Lever_16cm_til_servo_Q" AND NOT "Vent_ny_pall_16cm";
   IF "16cm_knapp_main_skap" THEN "16cm_pall_på_plass" := TRUE; END_IF;
   "Ventil_6_UT" := "Ved_hentPos16cm_fra_servo" AND NOT "C6_retur_set" AND "16cm_pall_på_plass";
   IF "C6_PlussPos_I" THEN
       "C6_retur_set" := TRUE;
       "Lever_8cm_til_servo_Q" := TRUE;
   END_IF;
   IF "C6_MinPos_I" THEN "C6_retur_set" := FALSE; END_IF;
   IF "C6_retur_set" THEN "16cm_pall_på_plass" := FALSE; END_IF;
   IF "Bekreftet_levert_pall_16cm_fra_servo" THEN
       "Lever_8cm_til_servo_Q" := FALSE;
       "Vent_ny_pall_16cm" := TRUE;
   END_IF;
   IF "16cm_knapp_main_skap" THEN "Vent_ny_pall_16cm" := FALSE; END_IF;
END_REGION
END_FUNCTION

ORGANIZATION_BLOCK "Main"   // OB1, LAD, ProgramCycle
{ S7_Optimized_Access := 'TRUE' }
VERSION : 0.1
   VAR_INPUT
      Initial_Call : Bool;
      Remanence : Bool;
   END_VAR
BEGIN

REGION Network 1
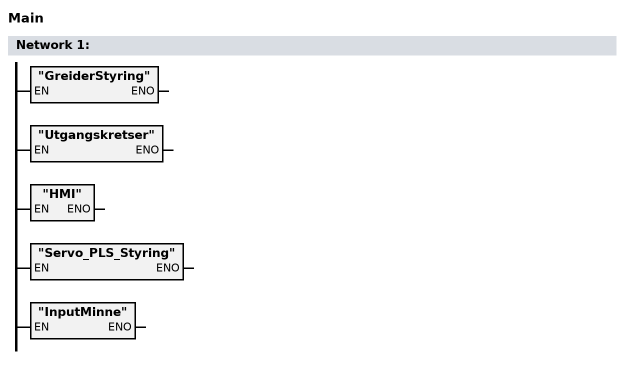
   RUNG wire#powerrail
      "GreiderStyring"()
   END_RUNG
   RUNG wire#powerrail
      "Utgangskretser"()
   END_RUNG
   RUNG wire#powerrail
      "HMI"()
   END_RUNG
   RUNG wire#powerrail
      "Servo_PLS_Styring"()
   END_RUNG
   RUNG wire#powerrail
      "InputMinne"()
   END_RUNG
   // the same network as SCL:
   "GreiderStyring"();
   "Utgangskretser"();
   "HMI"();
   "Servo_PLS_Styring"();
   "InputMinne"();
END_REGION
END_ORGANIZATION_BLOCK